TEXTLIST tl_OutputNames
  1 = 'Saida 01'
  2 = 'Saida 02'
  3 = 'Saida 03'
  4 = 'Saida 04'
  5 = 'Saida 05'
  6 = 'Saida 06'
  7 = 'Saida 07'
  8 = 'Saida 08'
   = ''
END_TEXTLIST

(* stored: Version 1.1.0.1
   TextList tl_OutputNames: Id {1a65c10c-185a-4017-9631-f6526ad8dc3a} *)
